FUNCTION_BLOCK FB_OnlyPVUpdate
VAR_INPUT
END_VAR
VAR_OUTPUT
END_VAR
VAR
	i: INT;
END_VAR

FOR i:=1 TO E_aAnalogInputIO_Index.E_PV_EPC_04 DO
	IF 0.0 < GVL_IO.aMaxValueController[i]  THEN		
		GVL_IO.aController_PV[i] := (GVL_IO.aAnalogInputIO[i] / GVL_CONSTANT.EL3064MaxValueH) * GVL_IO.aMaxValueController[i];
	END_IF
END_FOR

GVL_IO.aController_PV[E_aAnalogInputIO_Index.E_PV_Susceptor_Temp] := WORD_TO_REAL(GVL_IO.wE3508_PV);
GVL_IO.aController_PV[E_aAnalogInputIO_Index.E_PV_Reactor_Pressure] := WORD_TO_REAL(GVL_IO.wIqPlus_CDG2_PV);
GVL_IO.aController_PV[E_aAnalogInputIO_Index.E_PV_susceptorRotation] := GVL_IO.nRotation_Converted_PV;

END_FUNCTION_BLOCK

(* stored: Version 1.1.0.1, ProductVersion 3.1.4024.15
   POU FB_OnlyPVUpdate: Id {be8dea6c-02de-48fe-8c7a-f820ec1c1882}, SpecialFunc None *)
